(* IEC 61131-3 sources: Industry-PLC-LLM/data/PLCBEAD_repo/PLCBEAD_PLCEmbed-main/PLC-BEAD/Source/GEB/TIME_TO_TOD, 1 file *)

(* ---- TIME_TO_TOD.ST ---- *)
FUNCTION TIME_TO_TOD:UDINT

	VAR_INPUT
		IN :	TIME;
	END_VAR

	TIME_TO_TOD := DWORD_TO_UDINT(TIME_TO_DWORD(IN));
END_FUNCTION

PROGRAM program0
  VAR
	IN :	TIME;
    CEIL5_OUT : UDINT;
  END_VAR

  CEIL5_OUT := TIME_TO_TOD(IN);
END_PROGRAM
